FUNCTION_BLOCK RT_E_SELECT (* Selection between two events *)
  (* Standard: 61499-1; Classification: Event processing *)
  (* Version 0.0, 2008-07-10, 4DIAC-IDE, 4DIAC-Consortium *)
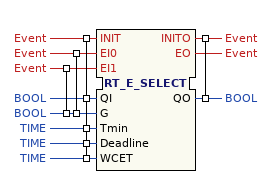
  EVENT_INPUT
    INIT WITH QI, Tmin, Deadline, WCET;
    EI0 WITH G; (* Input event,selected when G=0 *)
    EI1 WITH G; (* Input event,selected when G=1 *)
  END_EVENT
  EVENT_OUTPUT
    INITO WITH QO;
    EO; (* Output Event *)
  END_EVENT
  VAR_INPUT
    QI : BOOL;
    G : BOOL; (* Select EI0 when G=0,EI1 when G=1 *)
    Tmin : TIME;
    Deadline : TIME;
    WCET : TIME;
  END_VAR
  VAR_OUTPUT
    QO : BOOL;
  END_VAR
END_FUNCTION_BLOCK
